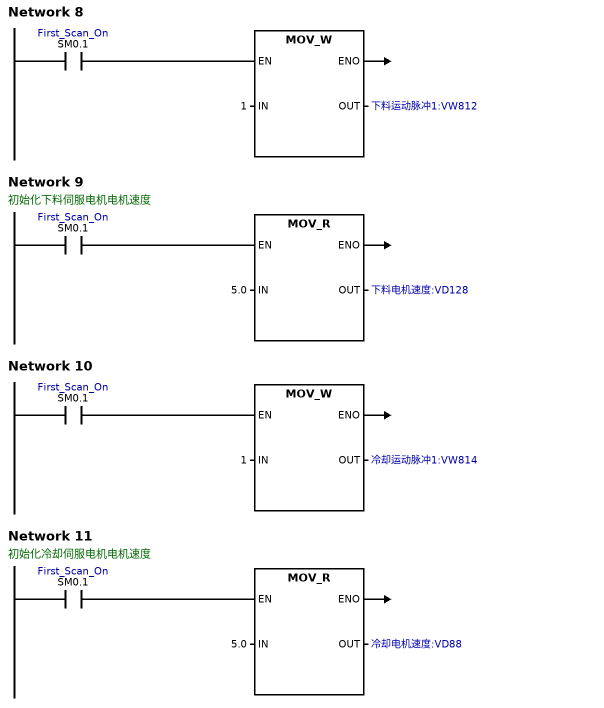
[picture p24: SBR20 networks 8-11]
Network 8
LD     First_Scan_On:SM0.1
MOVW   1, 下料运动脉冲1:VW812
Network 9
// 初始化下料伺服电机电机速度
LD     First_Scan_On:SM0.1
MOVR   5.0, 下料电机速度:VD128
Network 10
LD     First_Scan_On:SM0.1
MOVW   1, 冷却运动脉冲1:VW814
Network 11
// 初始化冷却伺服电机电机速度
LD     First_Scan_On:SM0.1
MOVR   5.0, 冷却电机速度:VD88
END_SUBROUTINE_BLOCK
